// TIA Portal V20 export
VAR_GLOBAL   // PLC tag table "MABS"
   "MABS_A1.9.1_IN" AT %I711.0 : "Global.IB_P01_02_03_in_64bytes_struct";
   "MABS_A1.9.1_Out" AT %Q633.0 : "Global.IB_P01_02_03_out_64bytes_struct";
   "MABS_A1.9.2_IN" AT %I775.0 : "Global.IB_P01_02_03_in_64bytes_struct";
   "MABS_A1.9.2_Out" AT %Q697.0 : "Global.IB_P01_02_03_out_64bytes_struct";
   "MABS_A1.6.1_IN" AT %I583.0 : "Global.IB_P01_02_03_in_64bytes_struct";
   "MABS_A1.6.1_Out" AT %Q505.0 : "Global.IB_P01_02_03_out_64bytes_struct";
   "MABS_A1.6.2_IN" AT %I647.0 : "Global.IB_P01_02_03_in_64bytes_struct";
   "MABS_A1.6.2_Out" AT %Q569.0 : "Global.IB_P01_02_03_out_64bytes_struct";
END_VAR
